{attribute 'GeneratedUsingTerminal: EP9128-0021-0018'}
{attribute addProperty BoxType "EP9128-0021-0018"}
{attribute addProperty Id "A_0013_EP9128_0021_0019A_0013_EP9128_0021_0019_0DE615A6579A_0010_EP9128_0021_0018_2_EP9128_1021EP9128_1FC0878B2A_0010_EP9128_0021_0018_3_EP9128_2021EP9128_1FC0878B2"}
{attribute addProperty CRC "3378115810"}
{attribute addProperty Size "583"}
TYPE A_0010_EP9128_0021_0018_C959F4E2 EXTENDS EP9128_1FC0878B :
STRUCT
	{attribute addProperty Name "A_0013_EP9128_0021_0019"}
	A_0013_EP9128_0021_0019 : A_0013_EP9128_0021_0019_0DE615A6;
	{attribute addProperty Name "A_0010_EP9128_0021_0018_2_EP9128_1021"}
	A_0010_EP9128_0021_0018_2_EP9128_1021 : EP9128_1FC0878B;
	{attribute addProperty Name "A_0010_EP9128_0021_0018_3_EP9128_2021"}
	A_0010_EP9128_0021_0018_3_EP9128_2021 : EP9128_1FC0878B;
END_STRUCT
END_TYPE

(* stored: Version 1.2.0.0, ProductVersion 3.1.4024.9
   DUT A_0010_EP9128_0021_0018_C959F4E2: Id {33d2452b-933c-4083-9f79-820a9042d9ec} *)
